{attribute addProperty BoxType "EPP2316-0003-0016"}
{attribute addProperty Id "Diag_InputAT %I*ARRAY[0 ..7] OF BOOL6480"}
{attribute addProperty CRC "265177097"}
{attribute addProperty SizeInBites "64"}
{attribute addProperty SizeInBytes "8"}
TYPE DIG_Diag_Inputs_AC4A9AF0 :
STRUCT
	{attribute addProperty Name "Diag_Input"}
	Diag_Input AT %I* : ARRAY[0 ..7] OF BOOL;
END_STRUCT
END_TYPE

(* stored: Version 1.2.0.0, ProductVersion 3.1.4024.9
   DUT DIG_Diag_Inputs_AC4A9AF0: Id {11ae34ef-e0e7-4100-a32a-2a2e546bf69f} *)
